// TIA Portal V15 program export: 0 tag tables, 0 data types, 0 data blocks, 6 code blocks (in call order from the OBs), 4 instance data blocks

ORGANIZATION_BLOCK "Main"   // OB1, LAD, ProgramCycle
TITLE = "Main Program Sweep (Cycle)"
{ S7_Optimized_Access := 'TRUE' }
// stored: SetENOAutomatically False
   VAR_INPUT
      Initial_Call : Bool;   // Initial call of this OB
      Remanence : Bool;   // =True, if remanent data are available
   END_VAR
BEGIN

REGION Network 1
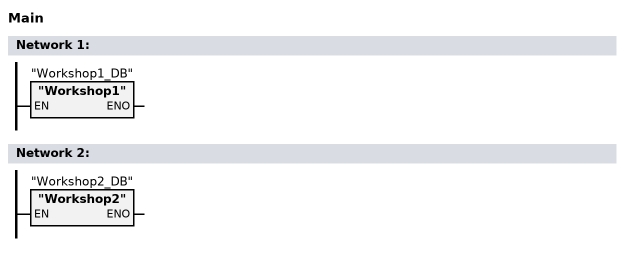
   RUNG wire#powerrail
      "Workshop1_DB"()
   END_RUNG
   // the same network as SCL:
   "Workshop1_DB"();   // "Workshop1"
END_REGION

REGION Network 2
   RUNG wire#powerrail
      "Workshop2_DB"()
   END_RUNG
   // the same network as SCL:
   "Workshop2_DB"();   // "Workshop2"
END_REGION
END_ORGANIZATION_BLOCK

FUNCTION_BLOCK "Workshop1"   // FB2, LAD
{ S7_Optimized_Access := 'TRUE' }
// stored: AutoNumber false, MemoryReserve 100, SetENOAutomatically False
BEGIN

REGION Network 1
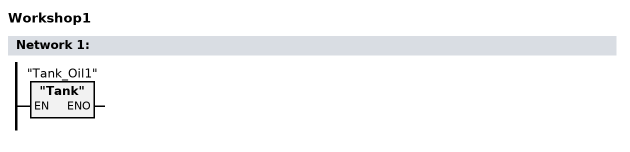
   RUNG wire#powerrail
      "Tank_Oil1"()
   END_RUNG
   // the same network as SCL:
   "Tank_Oil1"();   // "Tank"
END_REGION
END_FUNCTION_BLOCK

FUNCTION_BLOCK "Workshop2"   // FB3, LAD
{ S7_Optimized_Access := 'TRUE' }
// stored: MemoryReserve 100, SetENOAutomatically False
BEGIN

REGION Network 1
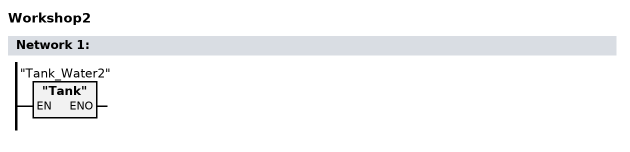
   RUNG wire#powerrail
      "Tank_Water2"()
   END_RUNG
   // the same network as SCL:
   "Tank_Water2"();   // "Tank"
END_REGION
END_FUNCTION_BLOCK

ORGANIZATION_BLOCK "Startup"   // OB100, LAD, Startup
TITLE = "Complete Restart"
{ S7_Optimized_Access := 'TRUE' }
// stored: SetENOAutomatically False
   VAR_INPUT
      LostRetentive : Bool;   // True if retentive data are lost
      LostRTC : Bool;   // True if date and time are lost
   END_VAR
BEGIN

REGION Network 1
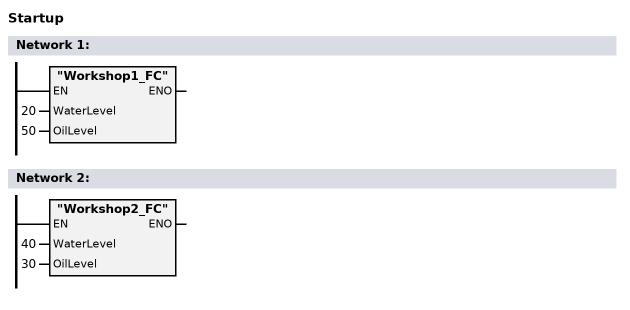
   RUNG wire#powerrail
      "Workshop1_FC"(WaterLevel := 20, OilLevel := 50)
   END_RUNG
   // the same network as SCL:
   "Workshop1_FC"(WaterLevel := 20, OilLevel := 50);
END_REGION

REGION Network 2
   RUNG wire#powerrail
      "Workshop2_FC"(WaterLevel := 40, OilLevel := 30)
   END_RUNG
   // the same network as SCL:
   "Workshop2_FC"(WaterLevel := 40, OilLevel := 30);
END_REGION
END_ORGANIZATION_BLOCK

FUNCTION "Workshop1_FC" : Void   // FC1, LAD
{ S7_Optimized_Access := 'TRUE' }
// stored: SetENOAutomatically False
   VAR_INPUT
      WaterLevel : Int;
      OilLevel : Int;
   END_VAR
BEGIN

REGION Network 1
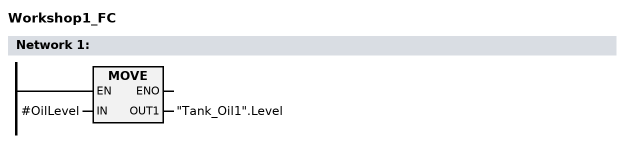
   RUNG wire#powerrail
      Move(in := #OilLevel, out1 => "Tank_Oil1".Level)
   END_RUNG
   // the same network as SCL:
   "Tank_Oil1".Level := #OilLevel;
END_REGION
END_FUNCTION

FUNCTION "Workshop2_FC" : Void   // FC2, LAD
{ S7_Optimized_Access := 'TRUE' }
// stored: SetENOAutomatically False
   VAR_INPUT
      WaterLevel : Int;
      OilLevel : Int;
   END_VAR
BEGIN

REGION Network 1
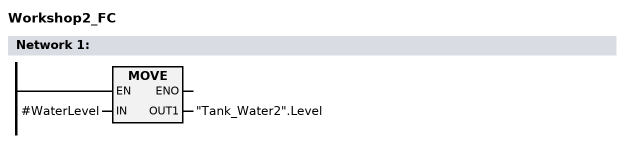
   RUNG wire#powerrail
      Move(in := #WaterLevel, out1 => "Tank_Water2".Level)
   END_RUNG
   // the same network as SCL:
   "Tank_Water2".Level := #WaterLevel;
END_REGION
END_FUNCTION

DATA_BLOCK "Workshop1_DB"   // DB3
{ S7_Optimized_Access := 'TRUE' }
// stored: InstanceOfName Workshop1
"Workshop1"
BEGIN
END_DATA_BLOCK

DATA_BLOCK "Workshop2_DB"   // DB6
{ S7_Optimized_Access := 'TRUE' }
// stored: InstanceOfName Workshop2
"Workshop2"
BEGIN
END_DATA_BLOCK

DATA_BLOCK "Tank_Oil1"   // DB2
{ S7_Optimized_Access := 'TRUE' }
// stored: InstanceOfName Tank
"Tank"
   // VAR
   //    Level : Int;
   // END_VAR
BEGIN
END_DATA_BLOCK

DATA_BLOCK "Tank_Water2"   // DB4
{ S7_Optimized_Access := 'TRUE' }
// stored: InstanceOfName Tank
"Tank"
   // VAR
   //    Level : Int;
   // END_VAR
BEGIN
END_DATA_BLOCK
